// TIA Portal V20 export
TYPE "LWONIK_typeFromSafetyDoorStatus"
// stored: Access Published
   STRUCT
      FdoorSwitchStatus : Struct
         maintDoorOpen : Bool;
         stack1NgBoxDoorOpen : Bool;
         stack2NgBoxDoorOpen : Bool;
         "transferP&PLDoorOpen" : Bool;
         "transferP&PRDoorOpen" : Bool;
         unloadingDoorOpen : Bool;
         ngBoxDoorOpen : Bool;
         laserMarkDoorClose : Bool;
         "h.PressDoorOpen" : Bool;
         sideTapingDoorOpen : Bool;
         topTapingDoorOpen : Bool;
      END_STRUCT;
      FdoorCoilStatus : Struct
         maintDoorUnlock : Bool;
         stack1NgBoxDoorUnlock : Bool;
         stack2NgBoxDoorUnlock : Bool;
         "transferP&PLDoorUnlock" : Bool;
         "transferP&PRDoorUnlock" : Bool;
         unloadingDoorUnlock : Bool;
         ngBoxDoorUnlock : Bool;
         laserMarkDoorUnlock : Bool;
         "h.PressDoorUnlock" : Bool;
         sideTapingDoorUnlock : Bool;
         topTapingDoorUnlock : Bool;
      END_STRUCT;
   END_STRUCT;
END_TYPE
